TYPE "UDT_TrackingReport_HMI_OP1"
VERSION : 0.1
   STRUCT
      ClearReport : Bool;
      PosInx_HMI : Int;
      PageNo : Int;
      RowIndex : Array[0..9] of Int;
      TrackingReport { S7_SetPoint := 'False'} : Array[0..9] of "UDT_TrackingReport_OP01";
   END_STRUCT;

END_TYPE

